// TIA Portal V17 export
// export: Created 2026-10-01T22:10:27.570325Z, ExportSetting WithDefaults, DisplayName Totally Integrated Automation Portal, DisplayVersion V17, DisplayName TIA Portal Openness, DisplayVersion V17, DisplayName TIA Portal Version Control Interface, DisplayVersion V17, DisplayName SINAMICS Startdrive Advanced, DisplayVersion V17, DisplayName SINAMICS Startdrive G130, G150, S120, S150, SINAMICS MV, G220, S200, S210, DisplayVersion V17, DisplayName SINAMICS Startdrive G110M, G120, G120C, G120D, G120P, G115D, DisplayVersion V17, DisplayName STEP 7 Professional, DisplayVersion V17, DisplayName STEP 7 Safety, DisplayVersion V17, DisplayName WinCC Basic/Comfort/Advanced, DisplayVersion V17, DisplayName WinCC Unified, DisplayVersion V17
FUNCTION_BLOCK "ZZ_LadTest_Sys"   // FB32, LAD
{ S7_Optimized_Access := 'TRUE' }
VERSION : 0.1
// stored: AutoNumber true, IsIECCheckEnabled false, IsRetainMemResEnabled false, MemoryReserve 100, SetENOAutomatically false, UDAEnableTagReadback false
   VAR_INPUT
      Go : Bool;
   END_VAR
   VAR
      "Dt" : DTL;
      Err : Int;
   END_VAR
BEGIN

REGION Network 1
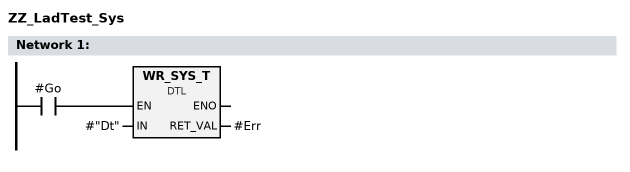
   RUNG wire#powerrail
      Contact( #Go )
      { S7_Templates := "date_type := DTL" } WR_SYS_T(IN := #"Dt", RET_VAL => #Err)
   END_RUNG
   // the same network as SCL:
   IF #Go THEN #Err := WR_SYS_T(IN := #"Dt"); END_IF;
END_REGION
END_FUNCTION_BLOCK
